FUNCTION_BLOCK FB_StringManager

VAR
	_workString : T_MaxString;
END_VAR

METHOD Append : REFERENCE TO FB_StringManager
VAR_INPUT
	Text : T_MaxString;
END_VAR
_workString:= Concat(_workString,text);
Append ref= THIS^;
END_METHOD

METHOD Reset : REFERENCE TO FB_StringManager
VAR_INPUT
END_VAR
_workString:='';
Reset ref= THIS^;
END_METHOD

METHOD ToString : T_MaxString
VAR_INPUT
END_VAR
ToString := _workString;
END_METHOD

END_FUNCTION_BLOCK

(* stored: Version 1.1.0.1, ProductVersion 3.1.4024.12
   POU FB_StringManager: Id {18fc62f0-9bc4-4d7b-b56a-a97b69b2ef18}, SpecialFunc None
   Method Append: Id {7d3e3917-3482-48d8-8b88-9a05889006f7}
   Method Reset: Id {bcf8c3b8-b4fb-4db4-8dd5-3556c56a1691}
   Method ToString: Id {63e51bb5-494a-4223-b8ac-117dd087815a} *)
